// TIA Portal V16 export
// export: Created 2021-09-16T19:23:53.0393489Z, ExportSetting WithDefaults, DisplayName Totally Integrated Automation Portal, DisplayVersion V16 Update 4, DisplayName TIA Portal Version Control Interface, DisplayVersion V16 Update 2, DisplayName TIA Portal Openness, DisplayVersion V16 Update 4, DisplayName STEP 7 Professional, DisplayVersion V16 Update 4, DisplayName STEP 7 Safety, DisplayVersion V16, DisplayName WinCC Advanced, DisplayVersion V16 Update 4
VAR_GLOBAL   // PLC tag table "Default tag table"
   estop_clear AT %I0.0 : Bool;   //    {ExternalAccessible false, ExternalVisible false, ExternalWritable false}
   interlock AT %Q0.0 : Bool;   //    {ExternalAccessible false, ExternalVisible false, ExternalWritable false}
   reset AT %I0.1 : Bool;   //    {ExternalAccessible false, ExternalVisible false, ExternalWritable false}
END_VAR
